Staubli VAL3: RefreshList.pgx

program RefreshList()
  local num l_ni
begin
  if bListRefresh
    for l_ni=0 to nSize-1
      sList[l_ni]=toString("",l_ni+1)+"点"
    endFor
  endIf

end
